(* CODESYS project gp60t.project

Project tree, tasks and I/O mapping:
  Device : SPK1xx[M01], Production association OWEN, order no. 1, version 3.5.17.31
    application Application
      libraries: Standard, * (System); Util, * (System); CAA DTUtil Extern, * (CAA Technical Workgroup); VisuDialogs, * (System); Standard64, * (System); SysCom, * (System); CmpBitmapPool, * (System); CmpSysExec, 3.5.17.31 (Production association OWEN); Visu Utils, 4.1.0.0 (System); OwenStringUtils, 3.5.4.7 (Production association OWEN); CAA File, 3.5.17.0 (CAA Technical Workgroup); VisuKeyboard_En-Ru, 1.3.0.0 (PC Prolog)
      task VISU_TASK (cyclic, interval 100 ms, priority 10) calls VisuElems.Visu_Prg
      task MainTask (cyclic, interval 50 ms, priority 2) calls Main
      task AlarmManagerTask (cyclic, interval 1030 ms, priority 15) calls AlarmManager.Alarm_Prg
      POUs/
        gp/
          program CalcTech [ST]: remap, roundTo, DEGR_TO_RAD, fcFindOfEquip, fcFindOfSup, remap_1, RAD_TO_DEGR, ACT_AUTO_MATRIX, pickRangeNumber, ACT_GEOMETRY, pickRangeNumberLinear, ACT_ANGLE_MACHINE, ceil, ACT_MATRIX, ACT_ELASTIC_MOVE
          Data_types/
            data type warning
            data type recType
            data type SupportType
            data type Ustav
            data type test
            data type Union_Real
            data type dataBase
            data type OperTime
            data type FindOfEq
            data type recType2
            data type Equipment
            data type middle_line
            data type Steel
            data type Accept_struct
            data type SupportType2
          program Actuators [ST]: ACT_INPUT
          function block fbAlrmMove [ST]
          program recipes [ST]: addData, DelData, AddEquip, DelScrew, DelSteel, setScrew, AddScrew, setData, getSteel, DelEquip, getData, getSupport, AddSupport, findName, setSupport, getEquip, addSteel, setEquip, DelSupport, getScrew, setSteel
          function block fbSensor [ST]
          program Main [ST]: ACT_INPUT
          program Visu_var [ST]
          function block fbControl_sys [ST]
          function block Operating_time_v1 [ST]
          function block fbCylinder [ST]
          function block fbActuator [ST]
          function block simulateMove [ST]
        _System/
          function block waitingScreen [ST]
          function block MessageEx [ST]
          function block TimeToString [ST]
          function WhatTime [ST]
          TimeSetup/
            program TimeSetup [ST]
            function block RealTimeClock4 [ST]
            function Day2weekDay [ST]
            function block UpdateUint [ST]
          function block ConvToVolt [CFC]
          function fcSortInt [ST]
          function block RangeConvert [ST]
          function block simpleSPAD [ST]
          function getEquipKeypad [ST]
          function WhatCycleTime [ST]
          function dword2real [ST]
      RecipeManager
        recipe definition EquipGroup: arEquip[0].name : WSTRING(20); arEquip[0].place : WSTRING(10); arEquip[1].name : WSTRING(20); arEquip[1].place : WSTRING(10); arEquip[2].name : WSTRING(20); arEquip[2].place : WSTRING(10); arEquip[3].name : WSTRING(20); arEquip[3].place : WSTRING(10); arEquip[4].name : WSTRING(20); arEquip[4].place : WSTRING(10); arEquip[5].name : WSTRING(20); arEquip[5].place : WSTRING(10); arEquip[6].name : WSTRING(20); arEquip[6].place : WSTRING(10); arEquip[7].name : WSTRING(20); arEquip[7].place : WSTRING(10); arEquip[8].name : WSTRING(20); arEquip[8].place : WSTRING(10); arEquip[9].name : WSTRING(20); arEquip[9].place : WSTRING(10); arEquip[10].name : WSTRING(20); arEquip[10].place : WSTRING(10); arEquip[11].name : WSTRING(20); arEquip[11].place : WSTRING(10); arEquip[12].name : WSTRING(20); arEquip[12].place : WSTRING(10); arEquip[13].name : WSTRING(20); arEquip[13].place : WSTRING(10); arEquip[14].name : WSTRING(20); arEquip[14].place : WSTRING(10); arEquip[15].name : WSTRING(20); arEquip[15].place : WSTRING(10); arEquip[16].name : WSTRING(20); arEquip[16].place : WSTRING(10); arEquip[17].name : WSTRING(20); arEquip[17].place : WSTRING(10); arEquip[18].name : WSTRING(20); arEquip[18].place : WSTRING(10); arEquip[19].name : WSTRING(20); arEquip[19].place : WSTRING(10); arEquip[20].name : WSTRING(20); arEquip[20].place : WSTRING(10); arEquip[21].name : WSTRING(20); arEquip[21].place : WSTRING(10); arEquip[22].name : WSTRING(20); arEquip[22].place : WSTRING(10); arEquip[23].name : WSTRING(20); arEquip[23].place : WSTRING(10); arEquip[24].name : WSTRING(20); arEquip[24].place : WSTRING(10); arEquip[25].name : WSTRING(20); arEquip[25].place : WSTRING(10); arEquip[26].name : WSTRING(20); arEquip[26].place : WSTRING(10); arEquip[27].name : WSTRING(20); arEquip[27].place : WSTRING(10); arEquip[28].name : WSTRING(20); arEquip[28].place : WSTRING(10); arEquip[29].name : WSTRING(20); arEquip[29].place : WSTRING(10); arEquip[30].name : WSTRING(20); arEquip[30].place : WSTRING(10); arEquip[31].name : WSTRING(20); arEquip[31].place : WSTRING(10); arEquip[32].name : WSTRING(20); arEquip[32].place : WSTRING(10); arEquip[33].name : WSTRING(20); arEquip[33].place : WSTRING(10); arEquip[34].name : WSTRING(20); arEquip[34].place : WSTRING(10); arEquip[35].name : WSTRING(20); arEquip[35].place : WSTRING(10); arEquip[36].name : WSTRING(20); arEquip[36].place : WSTRING(10); arEquip[37].name : WSTRING(20); arEquip[37].place : WSTRING(10); arEquip[38].name : WSTRING(20); arEquip[38].place : WSTRING(10); arEquip[39].name : WSTRING(20); arEquip[39].place : WSTRING(10); arEquip[40].name : WSTRING(20); arEquip[40].place : WSTRING(10); arEquip[41].name : WSTRING(20); arEquip[41].place : WSTRING(10); arEquip[42].name : WSTRING(20); arEquip[42].place : WSTRING(10); arEquip[43].name : WSTRING(20); arEquip[43].place : WSTRING(10); arEquip[44].name : WSTRING(20); arEquip[44].place : WSTRING(10); arEquip[45].name : WSTRING(20); arEquip[45].place : WSTRING(10); arEquip[46].name : WSTRING(20); arEquip[46].place : WSTRING(10); arEquip[47].name : WSTRING(20); arEquip[47].place : WSTRING(10); arEquip[48].name : WSTRING(20); arEquip[48].place : WSTRING(10); arEquip[49].name : WSTRING(20); arEquip[49].place : WSTRING(10); arEquip[50].name : WSTRING(20); arEquip[50].place : WSTRING(10); arEquip[51].name : WSTRING(20); arEquip[51].place : WSTRING(10); arEquip[52].name : WSTRING(20); arEquip[52].place : WSTRING(10); arEquip[53].name : WSTRING(20); arEquip[53].place : WSTRING(10); arEquip[54].name : WSTRING(20); arEquip[54].place : WSTRING(10); arEquip[55].name : WSTRING(20); arEquip[55].place : WSTRING(10); arEquip[56].name : WSTRING(20); arEquip[56].place : WSTRING(10); arEquip[57].name : WSTRING(20); arEquip[57].place : WSTRING(10); arEquip[58].name : WSTRING(20); arEquip[58].place : WSTRING(10); arEquip[59].name : WSTRING(20); arEquip[59].place : WSTRING(10); arEquip[60].name : WSTRING(20); arEquip[60].place : WSTRING(10); arEquip[61].name : WSTRING(20); arEquip[61].place : WSTRING(10); arEquip[62].name : WSTRING(20); arEquip[62].place : WSTRING(10); arEquip[63].name : WSTRING(20); arEquip[63].place : WSTRING(10); arEquip[64].name : WSTRING(20); arEquip[64].place : WSTRING(10); arEquip[65].name : WSTRING(20); arEquip[65].place : WSTRING(10); arEquip[66].name : WSTRING(20); arEquip[66].place : WSTRING(10); arEquip[67].name : WSTRING(20); arEquip[67].place : WSTRING(10); arEquip[68].name : WSTRING(20); arEquip[68].place : WSTRING(10); arEquip[69].name : WSTRING(20); arEquip[69].place : WSTRING(10); arEquip[70].name : WSTRING(20); arEquip[70].place : WSTRING(10); arEquip[71].name : WSTRING(20); arEquip[71].place : WSTRING(10); arEquip[72].name : WSTRING(20); arEquip[72].place : WSTRING(10); arEquip[73].name : WSTRING(20); arEquip[73].place : WSTRING(10); arEquip[74].name : WSTRING(20); arEquip[74].place : WSTRING(10); arEquip[75].name : WSTRING(20); arEquip[75].place : WSTRING(10); arEquip[76].name : WSTRING(20); arEquip[76].place : WSTRING(10); arEquip[77].name : WSTRING(20); arEquip[77].place : WSTRING(10); arEquip[78].name : WSTRING(20); arEquip[78].place : WSTRING(10); arEquip[79].name : WSTRING(20); arEquip[79].place : WSTRING(10); arEquip[80].name : WSTRING(20); arEquip[80].place : WSTRING(10); arEquip[81].name : WSTRING(20); arEquip[81].place : WSTRING(10); arEquip[82].name : WSTRING(20); arEquip[82].place : WSTRING(10); arEquip[83].name : WSTRING(20); arEquip[83].place : WSTRING(10); arEquip[84].name : WSTRING(20); arEquip[84].place : WSTRING(10); arEquip[85].name : WSTRING(20); arEquip[85].place : WSTRING(10); arEquip[86].name : WSTRING(20); arEquip[86].place : WSTRING(10); arEquip[87].name : WSTRING(20); arEquip[87].place : WSTRING(10); arEquip[88].name : WSTRING(20); arEquip[88].place : WSTRING(10); arEquip[89].name : WSTRING(20); arEquip[89].place : WSTRING(10); arEquip[90].name : WSTRING(20); arEquip[90].place : WSTRING(10); arEquip[91].name : WSTRING(20); arEquip[91].place : WSTRING(10); arEquip[92].name : WSTRING(20); arEquip[92].place : WSTRING(10); arEquip[93].name : WSTRING(20); arEquip[93].place : WSTRING(10); arEquip[94].name : WSTRING(20); arEquip[94].place : WSTRING(10); arEquip[95].name : WSTRING(20); arEquip[95].place : WSTRING(10); arEquip[96].name : WSTRING(20); arEquip[96].place : WSTRING(10); arEquip[97].name : WSTRING(20); arEquip[97].place : WSTRING(10); arEquip[98].name : WSTRING(20); arEquip[98].place : WSTRING(10); arEquip[99].name : WSTRING(20); arEquip[99].place : WSTRING(10); arEquip[100].name : WSTRING(20); arEquip[100].place : WSTRING(10)
        recipe definition SteelGroup: arSteel[0].name : WSTRING(20); arSteel[0].t : DINT; arSteel[1].name : WSTRING(20); arSteel[1].t : DINT; arSteel[2].name : WSTRING(20); arSteel[2].t : DINT; arSteel[3].name : WSTRING(20); arSteel[3].t : DINT; arSteel[4].name : WSTRING(20); arSteel[4].t : DINT; arSteel[5].name : WSTRING(20); arSteel[5].t : DINT; arSteel[6].name : WSTRING(20); arSteel[6].t : DINT; arSteel[7].name : WSTRING(20); arSteel[7].t : DINT; arSteel[8].name : WSTRING(20); arSteel[8].t : DINT; arSteel[9].name : WSTRING(20); arSteel[9].t : DINT; arSteel[10].name : WSTRING(20); arSteel[10].t : DINT; arSteel[11].name : WSTRING(20); arSteel[11].t : DINT; arSteel[12].name : WSTRING(20); arSteel[12].t : DINT; arSteel[13].name : WSTRING(20); arSteel[13].t : DINT; arSteel[14].name : WSTRING(20); arSteel[14].t : DINT; arSteel[15].name : WSTRING(20); arSteel[15].t : DINT; arSteel[16].name : WSTRING(20); arSteel[16].t : DINT; arSteel[17].name : WSTRING(20); arSteel[17].t : DINT; arSteel[18].name : WSTRING(20); arSteel[18].t : DINT; arSteel[19].name : WSTRING(20); arSteel[19].t : DINT; arSteel[20].name : WSTRING(20); arSteel[20].t : DINT; arSteel[21].name : WSTRING(20); arSteel[21].t : DINT; arSteel[22].name : WSTRING(20); arSteel[22].t : DINT; arSteel[23].name : WSTRING(20); arSteel[23].t : DINT; arSteel[24].name : WSTRING(20); arSteel[24].t : DINT; arSteel[25].name : WSTRING(20); arSteel[25].t : DINT; arSteel[26].name : WSTRING(20); arSteel[26].t : DINT; arSteel[27].name : WSTRING(20); arSteel[27].t : DINT; arSteel[28].name : WSTRING(20); arSteel[28].t : DINT; arSteel[29].name : WSTRING(20); arSteel[29].t : DINT; arSteel[30].name : WSTRING(20); arSteel[30].t : DINT; arSteel[31].name : WSTRING(20); arSteel[31].t : DINT; arSteel[32].name : WSTRING(20); arSteel[32].t : DINT; arSteel[33].name : WSTRING(20); arSteel[33].t : DINT; arSteel[34].name : WSTRING(20); arSteel[34].t : DINT; arSteel[35].name : WSTRING(20); arSteel[35].t : DINT; arSteel[36].name : WSTRING(20); arSteel[36].t : DINT; arSteel[37].name : WSTRING(20); arSteel[37].t : DINT; arSteel[38].name : WSTRING(20); arSteel[38].t : DINT; arSteel[39].name : WSTRING(20); arSteel[39].t : DINT; arSteel[40].name : WSTRING(20); arSteel[40].t : DINT; arSteel[41].name : WSTRING(20); arSteel[41].t : DINT; arSteel[42].name : WSTRING(20); arSteel[42].t : DINT; arSteel[43].name : WSTRING(20); arSteel[43].t : DINT; arSteel[44].name : WSTRING(20); arSteel[44].t : DINT; arSteel[45].name : WSTRING(20); arSteel[45].t : DINT; arSteel[46].name : WSTRING(20); arSteel[46].t : DINT; arSteel[47].name : WSTRING(20); arSteel[47].t : DINT; arSteel[48].name : WSTRING(20); arSteel[48].t : DINT; arSteel[49].name : WSTRING(20); arSteel[49].t : DINT; arSteel[50].name : WSTRING(20); arSteel[50].t : DINT
        recipe definition SupGroup: arSupports[0].arLength[0] : INT; arSupports[0].arLength[1] : INT; arSupports[0].name : WSTRING(20); arSupports[1].arLength[0] : INT; arSupports[1].arLength[1] : INT; arSupports[1].name : WSTRING(20); arSupports[2].arLength[0] : INT; arSupports[2].arLength[1] : INT; arSupports[2].name : WSTRING(20); arSupports[3].arLength[0] : INT; arSupports[3].arLength[1] : INT; arSupports[3].name : WSTRING(20); arSupports[4].arLength[0] : INT; arSupports[4].arLength[1] : INT; arSupports[4].name : WSTRING(20); arSupports[5].arLength[0] : INT; arSupports[5].arLength[1] : INT; arSupports[5].name : WSTRING(20); arSupports[6].arLength[0] : INT; arSupports[6].arLength[1] : INT; arSupports[6].name : WSTRING(20); arSupports[7].arLength[0] : INT; arSupports[7].arLength[1] : INT; arSupports[7].name : WSTRING(20); arSupports[8].arLength[0] : INT; arSupports[8].arLength[1] : INT; arSupports[8].name : WSTRING(20); arSupports[9].arLength[0] : INT; arSupports[9].arLength[1] : INT; arSupports[9].name : WSTRING(20); arSupports[10].arLength[0] : INT; arSupports[10].arLength[1] : INT; arSupports[10].name : WSTRING(20); arSupports[11].arLength[0] : INT; arSupports[11].arLength[1] : INT; arSupports[11].name : WSTRING(20); arSupports[12].arLength[0] : INT; arSupports[12].arLength[1] : INT; arSupports[12].name : WSTRING(20); arSupports[13].arLength[0] : INT; arSupports[13].arLength[1] : INT; arSupports[13].name : WSTRING(20); arSupports[14].arLength[0] : INT; arSupports[14].arLength[1] : INT; arSupports[14].name : WSTRING(20); arSupports[15].arLength[0] : INT; arSupports[15].arLength[1] : INT; arSupports[15].name : WSTRING(20); arSupports[16].arLength[0] : INT; arSupports[16].arLength[1] : INT; arSupports[16].name : WSTRING(20); arSupports[17].arLength[0] : INT; arSupports[17].arLength[1] : INT; arSupports[17].name : WSTRING(20); arSupports[18].arLength[0] : INT; arSupports[18].arLength[1] : INT; arSupports[18].name : WSTRING(20); arSupports[19].arLength[0] : INT; arSupports[19].arLength[1] : INT; arSupports[19].name : WSTRING(20); arSupports[20].arLength[0] : INT; arSupports[20].arLength[1] : INT; arSupports[20].name : WSTRING(20); arSupports[21].arLength[0] : INT; arSupports[21].arLength[1] : INT; arSupports[21].name : WSTRING(20); arSupports[22].arLength[0] : INT; arSupports[22].arLength[1] : INT; arSupports[22].name : WSTRING(20); arSupports[23].arLength[0] : INT; arSupports[23].arLength[1] : INT; arSupports[23].name : WSTRING(20); arSupports[24].arLength[0] : INT; arSupports[24].arLength[1] : INT; arSupports[24].name : WSTRING(20); arSupports[25].arLength[0] : INT; arSupports[25].arLength[1] : INT; arSupports[25].name : WSTRING(20); arSupports[26].arLength[0] : INT; arSupports[26].arLength[1] : INT; arSupports[26].name : WSTRING(20); arSupports[27].arLength[0] : INT; arSupports[27].arLength[1] : INT; arSupports[27].name : WSTRING(20); arSupports[28].arLength[0] : INT; arSupports[28].arLength[1] : INT; arSupports[28].name : WSTRING(20); arSupports[29].arLength[0] : INT; arSupports[29].arLength[1] : INT; arSupports[29].name : WSTRING(20); arSupports[30].arLength[0] : INT; arSupports[30].arLength[1] : INT; arSupports[30].name : WSTRING(20); arSupports[31].arLength[0] : INT; arSupports[31].arLength[1] : INT; arSupports[31].name : WSTRING(20); arSupports[32].arLength[0] : INT; arSupports[32].arLength[1] : INT; arSupports[32].name : WSTRING(20); arSupports[33].arLength[0] : INT; arSupports[33].arLength[1] : INT; arSupports[33].name : WSTRING(20); arSupports[34].arLength[0] : INT; arSupports[34].arLength[1] : INT; arSupports[34].name : WSTRING(20); arSupports[35].arLength[0] : INT; arSupports[35].arLength[1] : INT; arSupports[35].name : WSTRING(20); arSupports[36].arLength[0] : INT; arSupports[36].arLength[1] : INT; arSupports[36].name : WSTRING(20); arSupports[37].arLength[0] : INT; arSupports[37].arLength[1] : INT; arSupports[37].name : WSTRING(20); arSupports[38].arLength[0] : INT; arSupports[38].arLength[1] : INT; arSupports[38].name : WSTRING(20); arSupports[39].arLength[0] : INT; arSupports[39].arLength[1] : INT; arSupports[39].name : WSTRING(20); arSupports[40].arLength[0] : INT; arSupports[40].arLength[1] : INT; arSupports[40].name : WSTRING(20); arSupports[41].arLength[0] : INT; arSupports[41].arLength[1] : INT; arSupports[41].name : WSTRING(20); arSupports[42].arLength[0] : INT; arSupports[42].arLength[1] : INT; arSupports[42].name : WSTRING(20); arSupports[43].arLength[0] : INT; arSupports[43].arLength[1] : INT; arSupports[43].name : WSTRING(20); arSupports[44].arLength[0] : INT; arSupports[44].arLength[1] : INT; arSupports[44].name : WSTRING(20); arSupports[45].arLength[0] : INT; arSupports[45].arLength[1] : INT; arSupports[45].name : WSTRING(20); arSupports[46].arLength[0] : INT; arSupports[46].arLength[1] : INT; arSupports[46].name : WSTRING(20); arSupports[47].arLength[0] : INT; arSupports[47].arLength[1] : INT; arSupports[47].name : WSTRING(20); arSupports[48].arLength[0] : INT; arSupports[48].arLength[1] : INT; arSupports[48].name : WSTRING(20); arSupports[49].arLength[0] : INT; arSupports[49].arLength[1] : INT; arSupports[49].name : WSTRING(20); arSupports[50].arLength[0] : INT; arSupports[50].arLength[1] : INT; arSupports[50].name : WSTRING(20); arSupports[51].arLength[0] : INT; arSupports[51].arLength[1] : INT; arSupports[51].name : WSTRING(20); arSupports[52].arLength[0] : INT; arSupports[52].arLength[1] : INT; arSupports[52].name : WSTRING(20); arSupports[53].arLength[0] : INT; arSupports[53].arLength[1] : INT; arSupports[53].name : WSTRING(20); arSupports[54].arLength[0] : INT; arSupports[54].arLength[1] : INT; arSupports[54].name : WSTRING(20); arSupports[55].arLength[0] : INT; arSupports[55].arLength[1] : INT; arSupports[55].name : WSTRING(20); arSupports[56].arLength[0] : INT; arSupports[56].arLength[1] : INT; arSupports[56].name : WSTRING(20); arSupports[57].arLength[0] : INT; arSupports[57].arLength[1] : INT; arSupports[57].name : WSTRING(20); arSupports[58].arLength[0] : INT; arSupports[58].arLength[1] : INT; arSupports[58].name : WSTRING(20); arSupports[59].arLength[0] : INT; arSupports[59].arLength[1] : INT; arSupports[59].name : WSTRING(20); arSupports[60].arLength[0] : INT; arSupports[60].arLength[1] : INT; arSupports[60].name : WSTRING(20); arSupports[61].arLength[0] : INT; arSupports[61].arLength[1] : INT; arSupports[61].name : WSTRING(20); arSupports[62].arLength[0] : INT; arSupports[62].arLength[1] : INT; arSupports[62].name : WSTRING(20); arSupports[63].arLength[0] : INT; arSupports[63].arLength[1] : INT; arSupports[63].name : WSTRING(20); arSupports[64].arLength[0] : INT; arSupports[64].arLength[1] : INT; arSupports[64].name : WSTRING(20); arSupports[65].arLength[0] : INT; arSupports[65].arLength[1] : INT; arSupports[65].name : WSTRING(20); arSupports[66].arLength[0] : INT; arSupports[66].arLength[1] : INT; arSupports[66].name : WSTRING(20); arSupports[67].arLength[0] : INT; arSupports[67].arLength[1] : INT; arSupports[67].name : WSTRING(20); arSupports[68].arLength[0] : INT; arSupports[68].arLength[1] : INT; arSupports[68].name : WSTRING(20); arSupports[69].arLength[0] : INT; arSupports[69].arLength[1] : INT; arSupports[69].name : WSTRING(20); arSupports[70].arLength[0] : INT; arSupports[70].arLength[1] : INT; arSupports[70].name : WSTRING(20); arSupports[71].arLength[0] : INT; arSupports[71].arLength[1] : INT; arSupports[71].name : WSTRING(20); arSupports[72].arLength[0] : INT; arSupports[72].arLength[1] : INT; arSupports[72].name : WSTRING(20); arSupports[73].arLength[0] : INT; arSupports[73].arLength[1] : INT; arSupports[73].name : WSTRING(20); arSupports[74].arLength[0] : INT; arSupports[74].arLength[1] : INT; arSupports[74].name : WSTRING(20); arSupports[75].arLength[0] : INT; arSupports[75].arLength[1] : INT; arSupports[75].name : WSTRING(20); arSupports[76].arLength[0] : INT; arSupports[76].arLength[1] : INT; arSupports[76].name : WSTRING(20); arSupports[77].arLength[0] : INT; arSupports[77].arLength[1] : INT; arSupports[77].name : WSTRING(20); arSupports[78].arLength[0] : INT; arSupports[78].arLength[1] : INT; arSupports[78].name : WSTRING(20); arSupports[79].arLength[0] : INT; arSupports[79].arLength[1] : INT; arSupports[79].name : WSTRING(20); arSupports[80].arLength[0] : INT; arSupports[80].arLength[1] : INT; arSupports[80].name : WSTRING(20); arSupports[81].arLength[0] : INT; arSupports[81].arLength[1] : INT; arSupports[81].name : WSTRING(20); arSupports[82].arLength[0] : INT; arSupports[82].arLength[1] : INT; arSupports[82].name : WSTRING(20); arSupports[83].arLength[0] : INT; arSupports[83].arLength[1] : INT; arSupports[83].name : WSTRING(20); arSupports[84].arLength[0] : INT; arSupports[84].arLength[1] : INT; arSupports[84].name : WSTRING(20); arSupports[85].arLength[0] : INT; arSupports[85].arLength[1] : INT; arSupports[85].name : WSTRING(20); arSupports[86].arLength[0] : INT; arSupports[86].arLength[1] : INT; arSupports[86].name : WSTRING(20); arSupports[87].arLength[0] : INT; arSupports[87].arLength[1] : INT; arSupports[87].name : WSTRING(20); arSupports[88].arLength[0] : INT; arSupports[88].arLength[1] : INT; arSupports[88].name : WSTRING(20); arSupports[89].arLength[0] : INT; arSupports[89].arLength[1] : INT; arSupports[89].name : WSTRING(20); arSupports[90].arLength[0] : INT; arSupports[90].arLength[1] : INT; arSupports[90].name : WSTRING(20); arSupports[91].arLength[0] : INT; arSupports[91].arLength[1] : INT; arSupports[91].name : WSTRING(20); arSupports[92].arLength[0] : INT; arSupports[92].arLength[1] : INT; arSupports[92].name : WSTRING(20); arSupports[93].arLength[0] : INT; arSupports[93].arLength[1] : INT; arSupports[93].name : WSTRING(20); arSupports[94].arLength[0] : INT; arSupports[94].arLength[1] : INT; arSupports[94].name : WSTRING(20); arSupports[95].arLength[0] : INT; arSupports[95].arLength[1] : INT; arSupports[95].name : WSTRING(20); arSupports[96].arLength[0] : INT; arSupports[96].arLength[1] : INT; arSupports[96].name : WSTRING(20); arSupports[97].arLength[0] : INT; arSupports[97].arLength[1] : INT; arSupports[97].name : WSTRING(20); arSupports[98].arLength[0] : INT; arSupports[98].arLength[1] : INT; arSupports[98].name : WSTRING(20); arSupports[99].arLength[0] : INT; arSupports[99].arLength[1] : INT; arSupports[99].name : WSTRING(20); arSupports[100].arLength[0] : INT; arSupports[100].arLength[1] : INT; arSupports[100].name : WSTRING(20)
